Staubli VAL3: userPage.pjx

--- userPage.pjx ---
Parameters version=s7.5 stackSize=5000 millimeterUnit=true
Program file=changeTrsf.pgx
Program file=changeValue.pgx
Program file=clear.pgx
Program file=divideString.pgx
Program file=editNumField.pgx
Program file=findPos.pgx
Program file=getListPosition.pgx
Program file=getMenu.pgx
Program file=getView.pgx
Program file=insertDialog.pgx
Program file=isListEmpty.pgx
Program file=leftPos.pgx
Program file=listadd.pgx
Program file=listcreate.pgx
Program file=listcursor.pgx
Program file=listdel.pgx
Program file=listempty.pgx
Program file=listevent.pgx
Program file=listframe.pgx
Program file=listins.pgx
Program file=listredraw.pgx
Program file=listupdate.pgx
Program file=midPos.pgx
Program file=nullKey.pgx
Program file=numCopy.pgx
Program file=printScroll.pgx
Program file=questionDialog.pgx
Program file=read.pgx
Program file=rightPos.pgx
Program file=scroll.pgx
Program file=selectNewField.pgx
Program file=setCenter.pgx
Program file=setMenu.pgx
Program file=setSizeList.pgx
Program file=setView.pgx
Program file=showBoolStatus.pgx
Program file=strfill.pgx
Program file=strfillchr.pgx
Program file=stringCopy.pgx
Program file=stringToArray.pgx
Program file=stringToFxArray.pgx
Program file=strlength.pgx
Program file=timerDialog.pgx
Program file=type.pgx
Program file=typeCenter.pgx
Program file=typeLen.pgx
Program file=typeMenu.pgx
Program file=yes_no.pgx
Program file=yes_no_cancel.pgx
Data file=userPage.dtx

--- userPage.dtx ---
bool Show
bool bReadWrite = true
public bool bShowDialog
public bool bUseEscape
public bool bUseRefresh
public num nBottomX[2]
  [0] = 17
  [1] = 17
public num nBottomY = 11
num nFirst
num nKey
num nOffSet
num nOldValue[2]
  [0] = 200
  [1] = 200
public num nPage = 10
public num nTopX[2]
  [0] = 21
  [1] = 21
public num nTopY
public num nView
public string sItems = "home"
string sMessage[3]
  [0] = "VALPLAST QUITTING..."
  [1] = " "
  [2] = "PLEASE WAIT"
public string sTitle = "HOME"

--- changeTrsf.pgx ---
public program changeTrsf(trsf& x_tTrsf[], string x_sTitle, string x_sComment)
  local bool l_bRefresh
  local num l_nView
  local num l_nIndex
  local string l_sItem
  local trsf l_tTrsf
  local string l_sEvent
  local string l_sEmpty
  local num l_nAddon
begin
  //logMsg("[KERNEL] INTERFACE:PAGE changeTrsf "+x_sTitle)
  // INIT all
  l_bRefresh=false
  l_nIndex=0
  l_nView=0
  call setSizeList(19,0,19,8)
  call setView(false)
  l_tTrsf=x_tTrsf
  //release the button
  call nullKey(nKey)
  // set the frame
  do
    cls()
    call type(0,12,x_sComment)
    call typeMenu(8,"OK")
    call listcreate(x_sTitle)
    l_sItem=("coord  X > "+toString(".2",l_tTrsf.x))
    call listadd(l_sItem)
    l_sItem=("coord  Y > "+toString(".2",l_tTrsf.y))
    call listadd(l_sItem)
    l_sItem=("coord  Z > "+toString(".2",l_tTrsf.z))
    call listadd(l_sItem)
    l_sItem=("coord RX > "+toString(".2",l_tTrsf.rx))
    call listadd(l_sItem)
    l_sItem=("coord RY > "+toString(".2",l_tTrsf.ry))
    call listadd(l_sItem)
    l_sItem=("coord RZ > "+toString(".2",l_tTrsf.rz))
    call listadd(l_sItem)
    // show the list
    nView=l_nIndex
    call listupdate(l_nIndex-l_nView)
    do
      l_nView=nView
      nKey=get()
      //l_pPoint.trsf=l_tTrsf
      call listevent(nKey,l_nIndex,l_sEvent)
      switch nKey
        case 270
          //
          // clean the line
          call listcursor(nView,false)
          l_sEmpty=""
          switch l_nIndex
            case 0
              //  x-value
              call changeValue(l_tTrsf.x,0,0,10+40-nBottomX,nView+1,l_sEmpty)
            break
            case 1
              //  y-value
              call changeValue(l_tTrsf.y,0,0,10+40-nBottomX,nView+1,l_sEmpty)
            break
            case 2
              //  z-value
              call changeValue(l_tTrsf.z,0,0,10+40-nBottomX,nView+1,l_sEmpty)
            break
            case 3
              //  rx-value
              call changeValue(l_tTrsf.rx,0,0,10+40-nBottomX,nView+1,l_sEmpty)
            break
            case 4
              //  ry-value
              call changeValue(l_tTrsf.ry,0,0,10+40-nBottomX,nView+1,l_sEmpty)
            break
            case 5
              //  rz-value
              call changeValue(l_tTrsf.rz,0,0,10+40-nBottomX,nView+1,l_sEmpty)
            break
            case 6
              // addon
              l_nIndex=find(l_sEvent,">")
              call changeValue(l_nAddon,0,0,l_nIndex+1+2+nTopX,nView+nTopY+1,l_sEmpty)
            break
          endSwitch
          l_bRefresh=true
        break
        case 278
          // VALIDATE
          x_tTrsf=l_tTrsf
        break
      endSwitch
    until l_bRefresh==true or nKey==255 or nKey==278
    l_bRefresh=false
  until nKey==255 or nKey==278
  // check the key
  if nKey==278
    // validate
    x_tTrsf=l_tTrsf
  endIf
  // release the resource
  call nullKey(nKey)
end

--- changeValue.pgx ---
public program changeValue(num& x_nValue[], num x_nMin, num x_nMax, num x_nX, num x_nY, string& x_sItems[])
  local num l_nOldValue[2]
  local string l_sItem
  local string l_sMessage
  local bool l_bComma
  local string l_sEmpty
begin
  //---------------------------------
  // Staubli copyright 2005
  //                By toneage
  //[Public]-------------------------
  //
  // x_nValue:  num to change
  // x_nMax:    max value
  // x_nMin:    min value
  // x_nX:      X position
  // x_nY:      Y position
  // x_sItems   message
  //
  // look if the value is between max and min
  //
  if x_nMin>x_nMax
    return
  endIf
  //
  // print the line in white
  //
  // call listCleanLine()
  //
  call nullKey(nKey)
  l_nOldValue[1]=round(x_nValue)
  x_nValue=(round(x_nValue*100))/100
  l_nOldValue=x_nValue
  // check if is using the comma or not
  if l_nOldValue!=l_nOldValue[1]
    l_bComma=true
  else
    l_bComma=false
  endIf
  // start
  call clear(0,13)
  do
    if x_sItems==""
      //
      //  use the get num
      //
      if l_bComma
        call strfill(l_sEmpty,len(toString(".2",x_nValue)),l_sEmpty)
      else
        call strfill(l_sEmpty,len(toString("",x_nValue)),l_sEmpty)
      endIf
      call type(x_nX,x_nY,l_sEmpty)
      gotoxy(x_nX,x_nY)
      nKey=get(x_nValue)
      // check the comma again
      if round(x_nValue)!=x_nValue
        l_bComma=true
      endIf
      //
      // CHECK for MIN MAX VALUE
      //
      if x_nMax!=x_nMin or x_nMin!=0
        if x_nValue>x_nMax
          //
          // ask if you want to continue
          //
          popUpMsg("MAX: "+toString(".2",x_nMax))
          x_nValue=l_nOldValue
          //x_nValue=x_nMax
          nKey=-1
        else
          if x_nValue<x_nMin
            //
            popUpMsg("MIN: "+toString(".2",x_nMin))
            //x_nValue=x_nMin
            x_nValue=l_nOldValue
            nKey=-1
          endIf
        endIf
      endIf
      //
      // UPDATE THE VALUE
      //
      if l_bComma
        call type(x_nX,x_nY,toString(".2",x_nValue))
      else
        call type(x_nX,x_nY,toString("",x_nValue))
      endIf
    else
      //
      // STRING CHOICE
      //
      // show a list if there is the place
      call setSizeList(x_nX-1,max(0,x_nY-1),40-x_nX-1,min(13-x_nY,size(x_sItems)))
      call listcreate("")
      call listadd(x_sItems)
      call selectNewField(x_nValue,x_nValue,0)
      do
        nKey=get()
        call listevent(nKey,x_nValue,l_sItem)
      until nKey==270 or nKey==255
    endIf
  until nKey==270 or nKey==255
  if nKey==255
    bUseEscape=true
    x_nValue=l_nOldValue
    if x_sItems!=""
      x_sItems=x_sItems[l_nOldValue]
    endIf
  else
    bUseEscape=false
  endIf
end

--- clear.pgx ---
public program clear(num pX (dimensions=1), num pY (dimensions=1))
  local num i
  local num lLen
begin
  //---------------------------------
  //      C L E A R   L I N E
  //---------------------------------
  // Erase a pY line from the column
  // pX to end
  //
  //
  call typeLen(pX,pY," ",40-pX)
  gotoxy(pX,pY)
end

--- divideString.pgx ---
program divideString(string& x_sMsg[] (dimensions=1), num& x_nLine[] (dimensions=1))
  local string l_sCopyMsg
  local num l_nLength
  local string l_sSwap
  local num l_nFlag
  local num l_nTotalFlag
  local string l_sCR
  local num l_nPosCR
  local num i
begin
  //
  //  using:
  // x_sMessage->  the message you want print to video
  // x_nLine->     the number of the line that will be use
  //
  //
  // CARRIAGE RETURN
  l_sCR="#"
  x_nLine=0
  //length of a line for a message
  l_nLength=38
  // copy the msg
  l_sCopyMsg=x_sMsg
  // first case
  call findPos(l_sCopyMsg,l_sCR,l_nPosCR)
  if (getDisplayLen(l_sCopyMsg)>l_nLength-1) or (l_nPosCR!=-1)
    // compose the message
    do
      l_sSwap=l_sCopyMsg
      // set the x_sMsg
      if size(x_sMsg)-1<x_nLine
        append(x_sMsg)
      endIf
      call findPos(l_sCopyMsg,l_sCR,l_nPosCR)
      //
      if (getDisplayLen(l_sCopyMsg)>l_nLength-1 or (l_nPosCR!=-1)) and x_nLine<8
        // divide the string
        l_nTotalFlag=0
        call findPos(l_sCopyMsg,l_sCR,l_nPosCR)
        //
        // divide the string
        //
        if l_nPosCR!=-1 and l_nPosCR<l_nLength
          // CARRIAGE RETURN
          call leftPos(l_sCopyMsg,l_nPosCR,l_sSwap)
          //l_sSwap=left(l_sCopyMsg,l_nPosCR)
          call rightPos(l_sCopyMsg,getDisplayLen(l_sCopyMsg)-(l_nPosCR)-1,l_sCopyMsg)
          //l_sCopyMsg=right(l_sCopyMsg,len(l_sCopyMsg)-(l_nPosCR)-1)
          if getDisplayLen(l_sSwap)==0
            l_sSwap=" "
          endIf
        else
          //
          // search for the space then return
          //
          do
            call findPos(l_sSwap," ",l_nFlag)
            //l_nFlag=find(l_sSwap," ")
            if l_nFlag!=-1 and l_nFlag<=l_nLength
              //l_sSwap=right(l_sSwap,len(l_sSwap)-l_nFlag-1)
              call rightPos(l_sSwap,getDisplayLen(l_sSwap)-l_nFlag-1,l_sSwap)
              l_nTotalFlag=l_nTotalFlag+l_nFlag+1
            else
              if l_nTotalFlag==0 and (l_nFlag==-1 or l_nFlag>l_nLength)
                l_nFlag=-1
                l_nTotalFlag=38
              endIf
            endIf
          until l_nTotalFlag>=l_nLength+2 or l_nFlag==-1
          // NORMAL
          if l_nTotalFlag==0
            // FULL LINE
            call leftPos(l_sCopyMsg,l_nLength,l_sSwap)
            //l_sSwap=left(l_sCopyMsg,l_nLength)
            //l_sCopyMsg=right(l_sCopyMsg,len(l_sCopyMsg)-l_nLength)
            call rightPos(l_sCopyMsg,getDisplayLen(l_sCopyMsg)-l_nLength,l_sCopyMsg)
          else
            // DIVIDE IT
            call leftPos(l_sCopyMsg,l_nTotalFlag-l_nFlag-2,l_sSwap)
            //l_sSwap=left(l_sCopyMsg,l_nTotalFlag-l_nFlag-2)
            //l_sCopyMsg=right(l_sCopyMsg,len(l_sCopyMsg)-(l_nTotalFlag-l_nFlag-1))
            call rightPos(l_sCopyMsg,getDisplayLen(l_sCopyMsg)-(l_nTotalFlag-l_nFlag-1),l_sCopyMsg)
          endIf
        endIf
        // set the string
        x_sMsg[x_nLine]=l_sSwap
        x_nLine=x_nLine+1
      else
        // limit the string
        call rightPos(l_sSwap,l_nLength,x_sMsg[x_nLine])
        //x_sMsg[x_nLine]=right(l_sSwap,l_nLength)
        l_sSwap=""
      endIf
    until l_sSwap==""
  endIf
end

--- editNumField.pgx ---
public program editNumField(string x_sTitle, string& x_sItemName[], num& x_nItem[], num& x_nMin[], num& x_nMax[])
  local num j
  local num l_nSize
  local num l_nKey
  local string l_sEvent
  local num l_nIndex
  local num l_nField
  local string l_sItem
  local num i
  local string l_sEmpty
begin
  //
  // clear & copy
  //
  // nView=nFirst=0
  //call listempty()
  call numCopy(x_nItem,nOldValue)
  call numCopy(x_nItem,nOffSet)
  for j=0 to size(nOffSet)-1
    nOffSet[j]=0
  endFor
  // take the size
  l_nSize=size(x_nItem)-1
  // create the LIST
  call setSizeList(2,max((6-l_nSize/2)-2,2),34,min((l_nSize+1),8))
  call listcreate(x_sTitle)
  //
  // insert items
  //
  for j=0 to l_nSize
    l_sItem=x_sItemName[j]
    if l_sItem!=""
      call strlength(l_sItem,26)
      l_sItem=l_sItem+": "+toString(".1",x_nItem[j])
      call listadd(l_sItem)
      nOffSet[j]=nOffSet[max(j-1,0)]
    else
      nOffSet[j]=nOffSet[max(j-1,0)]+1
    endIf
  endFor
  // update the list
  call listupdate(0)
  do
    call clear(0,13)
    call typeMenu(8,"OK")
    l_nKey=get()
    call listevent(l_nKey,l_nIndex,l_sEvent)
    // use the offset
    i=l_nIndex+nOffSet[max(l_nIndex,0)]
    // on Enter Key
    if l_nKey==270
      call listcursor(l_nIndex,false)
      if size(x_nMin)==size(x_nItem)
        // use min and max
        l_sEmpty=""
        call changeValue(x_nItem[i],x_nMin[i],x_nMax[i],31,nView+nTopY+1,l_sEmpty)
      else
        call changeValue(x_nItem[i],x_nMin,x_nMax,31,nView+nTopY+1,l_sEmpty)
      endIf
      // UPDATE
      call listdel(l_nIndex)
      l_sItem=x_sItemName[i]
      call strlength(l_sItem,26)
      l_sItem=l_sItem+": "+toString(".1",x_nItem[i])
      call listins(l_sItem,l_nIndex)
      call listupdate(l_nIndex-nView)
    endIf
  until l_nKey==278 or l_nKey==255
  // escape use ?
  if l_nKey==255
    bUseEscape=true
    call numCopy(nOldValue,x_nItem)
  else
    bUseEscape=false
  endIf
  // exit
  call nullKey(l_nKey)
end

--- findPos.pgx ---
public program findPos(string x_sItem1 (dimensions=1), string x_sItem2 (dimensions=1), num& x_nPos[] (dimensions=1))
  local num l_nPos
begin
  // find the char using getDisplayLen
  l_nPos=find(x_sItem1,x_sItem2)
  if l_nPos!=-1
    x_nPos=getDisplayLen(left(x_sItem1,l_nPos))
  else
    x_nPos=-1
  endIf
end

--- getListPosition.pgx ---
public program getListPosition(num& x_nIndexX[] (dimensions=1), num& x_nIndexY[] (dimensions=1))
begin
  x_nIndexX=nTopX+1
  x_nIndexY=nFirst+nView+nTopY+1
end

--- getMenu.pgx ---
public program getMenu(string& x_sMenu[] (dimensions=1), bool& x_bUseMenu[] (dimensions=1))
// set the function button using the menu string
  local num i
begin
  //
  // STAUBLI Application
  // set the x_bUseMenu using the Menu
  // array string
  //
  for i=0 to (size(x_bUseMenu)-1)
    x_bUseMenu[i]=false
    if (size(x_sMenu)-1)>=i
      if x_sMenu[i]!=""
        // active the button
        x_bUseMenu[i]=true
      endIf
    endIf
  endFor
end

--- getView.pgx ---
public program getView(bool& x_bView[] (dimensions=1))
begin
  if nBottomX==38
    x_bView=true
  else
    x_bView=false
  endIf
end

--- insertDialog.pgx ---
public program insertDialog(string x_sMsg, num& x_nItem[], num x_nMin, num x_nMax)
  local num l_nStartLine
  local num l_nLine
  local num i
  local num l_nPX
  local num l_nPY
  local string l_sItem
  local string l_sMessage
  local string l_sEmpty
begin
  //
  // modify the x_sItem, using a min max range
  //
  if watch(bShowDialog==false,3)==false
    bShowDialog=false
    return
  else
    setMutex(bShowDialog)
    // clear the line
    call clear(0,13)
    // look for the comma
    if round(x_nItem)!=x_nItem
      l_sItem=toString(".2",x_nItem)
    else
      l_sItem=toString("",x_nItem)
    endIf
    // print the line
    l_sItem=x_sMsg+">"+l_sItem
    call stringCopy(l_sItem,sMessage)
    // divide the sentence
    call divideString(sMessage,l_nLine)
    l_nStartLine=round(5-l_nLine/2)
    // Start LINE
    call type(0,l_nStartLine-2,"┌──────────────────────────────────────┐")
    call type(0,l_nStartLine-1,"│                                      │")
    // write the message
    for i=0 to l_nLine
      //call type(,"                                      ")
      l_sMessage=sMessage[i]
      call typeCenter(i+l_nStartLine,l_sMessage,38,false)
      call type(0,l_nStartLine+i,"│"+l_sMessage+"│")
    endFor
    // end LINE
    call type(0,l_nStartLine+l_nLine+1,"│                                      │")
    call type(0,l_nStartLine+l_nLine+2,"└──────────────────────────────────────┘")
    l_nPX=find(l_sMessage,">")+2
    l_nPY=l_nStartLine+l_nLine
    // change the value
    call changeValue(x_nItem,x_nMin,x_nMax,l_nPX,l_nPY,l_sEmpty)
    //
    bShowDialog=false
    bUseRefresh=true
    //
  endIf
end

--- isListEmpty.pgx ---
public program isListEmpty(bool& x_bEmpty[] (dimensions=1))
begin
  if size(sItems)==1 and sItems[0]==""
    x_bEmpty=true
  else
    x_bEmpty=false
  endIf
end

--- leftPos.pgx ---
public program leftPos(string x_sItem (dimensions=1), num x_nLength (dimensions=1), string& x_sResult[] (dimensions=1))
  local num i
  local num l_nLength
  local string l_sItem
begin
  //
  l_sItem=x_sItem
  //
  if len(l_sItem)!=getDisplayLen(l_sItem) and x_nLength>0
    for i=0 to len(x_sItem)-1
      l_nLength=l_nLength+getDisplayLen(left(l_sItem,1))
      l_sItem=right(l_sItem,len(l_sItem)-1)
      if l_nLength==x_nLength
        x_sResult=left(x_sItem,i+1)
        return
      else
        if l_nLength>x_nLength
          x_sResult=left(x_sItem,i)
          return
        endIf
      endIf
    endFor
    // else
  endIf
  x_sResult=left(x_sItem,max(x_nLength,0))
  // endIf
end

--- listadd.pgx ---
public program listadd(string& x_sItems[] (dimensions=1))
  local num i
  local num l_nSize
begin
  //---------------------------------
  // insert x_sItems into the list
  //---------------------------------
  //
  // x_sItems:      Items to add
  //
  //---------------------------------
  // Staubli copyright 2005
  //                By toneage
  //[Public]-------------------------
  //
  //
  for i=0 to (size(x_sItems)-1)
    if (size(sItems)!=1 or sItems!="") and x_sItems[i]!=""
      insert(sItems[size(sItems)])
      insert(bReadWrite[size(bReadWrite)])
    endIf
    if x_sItems[i]!=""
      sItems[size(sItems)-1]=x_sItems[i]
      // for default the RW is true
      bReadWrite[size(bReadWrite)-1]=true
    endIf
  endFor
end

--- listcreate.pgx ---
public program listcreate(string x_sTitle)
begin
  //
  // Staubli Copyright 2003 07 31
  //
  sTitle=x_sTitle
  call listframe(sTitle,nTopX,nTopY,nBottomX,nBottomY)
  call listempty()

end

--- listcursor.pgx ---
public program listcursor(num pView (dimensions=1), bool pShow (dimensions=1))
  local num lX
  local num lY
  local string message
  local bool l_bEmpty
begin
  //
  // toneage Staubli Copyright 2005
  //
  call isListEmpty(l_bEmpty)
  if !l_bEmpty
    nView=pView
    lX=nTopX+1
    lY=nTopY+1+pView
    if (nView+nFirst)>(size(sItems)-1)
      call strfill(sItems[size(sItems)-1],nBottomX,message)
    else
      call strfill(sItems[max(0,nView+nFirst)],nBottomX,message)
    endIf
    gotoxy(lX,lY)
    if (pShow==true)
      setTextMode(1)
      put(message)
      setTextMode(0)
    else
      setTextMode(0)
      put(message)
    endIf
  endIf
end

--- listdel.pgx ---
public program listdel(num x_nIndex (dimensions=1))
  local num l_nSize
begin
  //
  // Staubli Copyright 2005 toneage
  //
  l_nSize=size(sItems)-1
  if ((x_nIndex>=0) and (x_nIndex<=l_nSize))
    if l_nSize>0
      delete(sItems[x_nIndex])
      delete(bReadWrite[x_nIndex])
    else
      sItems=""
      bReadWrite=true
    endIf
  endIf
end

--- listempty.pgx ---
public program listempty()
  local num lI
  local num lLen
  local string lRun[5]
  local num lRuni
begin
  //
  // Staubli Copyright 2003 06 20
  //
  lLen=size(sItems)-1
  for lI=0 to lLen
    if lI>0
      delete(sItems[0])
      delete(bReadWrite[0])
    endIf
  endFor
  sItems=""
  //
end

--- listevent.pgx ---
public program listevent(num pkey (dimensions=1), num& pIndex[] (dimensions=1), string& pItem[] (dimensions=1))
  local num lVal
  local num l_nSize
  local bool l_bEmpty
begin
  //
  // Toneage Staubli product
  //
  //
  // get the item in the list and scroll it
  //
  call isListEmpty(l_bEmpty)
  // not allowed negative value
  nView=max(0,nView)
  nFirst=max(0,nFirst)
  pIndex=max(0,pIndex)
  // look for the empty
  if !l_bEmpty
    l_nSize=size(sItems)-1
    // check the overFlow
    l_nSize=size(sItems)-1
    if (nFirst+nView>l_nSize)
      // reset the value
      nFirst=nView=0
    endIf
    // security...
    switch (pkey)
      //Up
      case 261
        if ((nView-1)>=0)
          // no need to scroll only change cursor position
          call listcursor(nView,false)
          nView=nView-1
          call listcursor(nView,true)
          // print the scroll
          //call printScroll()
        else
          if nView==0
            // scroll up
            if ((nFirst-1)>=0)
              nFirst=nFirst-1
              call listupdate(nFirst)
            else
              // go to the end
              if nView+nFirst!=l_nSize
                call listcursor(nView,false)
                call selectNewField(l_nSize,nFirst+nView,nView)
              endIf
            endIf
          endIf
        endIf
      break
      //Down
      case 266
        if ((nView+nFirst+1)<size(sItems))
          // no need to scroll only chenge cursor position
          if ((nView+1)<nBottomY)
            call listcursor(nView,false)
            nView=nView+1
            call listcursor(nView,true)
            // print the scroll
            //call printScroll()
          else
            // move UP
            nFirst=nFirst+1
            call listupdate(nFirst)
          endIf
        else
          // go to the top
          if !(nView==0 and nFirst==0)
            call listcursor(nView,false)
            nView=0
            call listupdate(0)
          endIf
        endIf
      break
      //Page Up
      case 262
        if !(nView==0 and nFirst==0)
          call listcursor(nView,false)
          if ((nFirst+nView-nBottomY)>=0)
            // move one page up
            call selectNewField(nFirst+nView-nBottomY,nFirst+nView,nView)
          else
            // go to home
            nView=0
            call listupdate(0)
          endIf
        endIf
      break
      //Page Down
      case 267
        if nView+nFirst!=l_nSize
          call listcursor(nView,false)
          if ((nView+nFirst+nBottomY)<size(sItems)-1)
            // move one page down
            call selectNewField(nFirst+nView+nBottomY,nFirst+nView,nView)
          else
            // go to the end
            call selectNewField(l_nSize,nFirst+nView,nView)
          endIf
        endIf
      break
      //End
      case 269
        if nView+nFirst!=l_nSize
          // move to end
          call listcursor(nView,false)
          call selectNewField(l_nSize,nFirst+nView,nView)
        endIf
      break
      //Home
      case 265
        if !(nView==0 and nFirst==0)
          // move to home
          call listcursor(nView,false)
          nView=0
          call listupdate(0)
        endIf
      break
      default
      break
    endSwitch
    pIndex=nFirst+nView
    pItem=sItems[pIndex]
    //
  else
    // reset the item
    pItem=""
    pIndex=0
  endIf
end

--- listframe.pgx ---
program listframe(string pTitle (dimensions=1), num pX (dimensions=1), num pY (dimensions=1), num pDx (dimensions=1), num pDy (dimensions=1))
  local num lDx
  local num lDy
  local num lI
  local num lJ
  local string lStr
  local string lStrLine
  local num lValue
begin
  //
  // Staubli Copyright 2003 06 20
  //
  lStrLine="─────────────────────────────────────────"
  lDx=pDx
  lDy=pDy
  //Top
  lStr="┌"+mid(lStrLine,lDx,0)+"┐"
  gotoxy(pX,pY)
  put(lStr)
  lValue=pX+2
  //Title
  if pTitle!=""
    call leftPos("┤"+pTitle+"│",lDx+1,pTitle)
    gotoxy(pX+lDx-getDisplayLen(pTitle)+2,pY)
    put(pTitle)
  endIf
  //Containt
  for lJ=1 to lDy
    lValue=pY+lJ
    lStr="│"
    gotoxy(pX,lValue)
    put(lStr)
    gotoxy(pX+lDx+1,lValue)
    put(lStr)
  endFor
  //Bottom
  lValue=pY+lJ
  lStr="└"+mid(lStrLine,lDx,0)+"┘"
  gotoxy(pX,lValue)
  put(lStr)
end

--- listins.pgx ---
public program listins(string& x_sItems[] (dimensions=1), num x_nPos (dimensions=1))
  local num i
  local num l_nSize
begin
  //
  // Staubli Copyright 2005
  //
  l_nSize=size(sItems)-1
  if ((x_nPos>=0) and (x_nPos<=l_nSize))
    for i=0 to (size(x_sItems)-1)
      if size(sItems)!=1 or sItems!=""
        insert(sItems[x_nPos+i])
        insert(bReadWrite[x_nPos+i])
      endIf
      sItems[x_nPos+i]=x_sItems[i]
      // for default the RW is true
      bReadWrite[x_nPos+i]=true
    endFor
  else
    call listadd(x_sItems)
  endIf
end

--- listredraw.pgx ---
public program listredraw(num pFirst (dimensions=1))
begin
  //
  // Staubli Copyright 2003 06 20
  //
  call listframe(sTitle,nTopX,nTopY,nBottomX,nBottomY)
  call listupdate(pFirst)
end

--- listupdate.pgx ---
public program listupdate(num pFirst)
  local num lI
  local num lLen
  local string lStr
  local string lStr2
  local num lValue
  local num lView
  local num lX
  local num lY
  local num l_nSize
  local bool l_bEmpty
begin
  //
  // insert into the box all the data
  //
  // to prevent a negative value
  if pFirst>0
    nFirst=pFirst
  else
    nFirst=0
  endIf
  // save the coordinate
  lValue=nBottomY-1
  // check the overFlow
  l_nSize=size(sItems)-1
  if (nFirst+nView>l_nSize)
    // reset the value
    nFirst=nView=0
  endIf
  lI=0
  // check the unKnow poblem
  if l_nSize<lValue
    if nFirst!=0
      nView=nView+nFirst
      nFirst=0
    endIf
  endIf
  do
    lX=nTopX+1
    lY=nBottomY+lI-1
    lY=nTopY+lI+1
    lLen=nBottomX
    if ((lI+nFirst)<size(sItems))
      // print the item
      if (l_nSize>=0)
        lStr=mid(sItems[(lI+nFirst)],lLen,0)
      endIf
    else
      // print the blank line
      lStr="                                        "
    endIf
    // fill the line
    call strfill(lStr,lLen,lStr2)
    gotoxy(lX,lY)
    put(lStr2)
    lI=lI+1
  until (lI>lValue)
  // underlien the actual line
  call isListEmpty(l_bEmpty)
  if !l_bEmpty
    call listcursor(nView,true)
  else
    call listcursor(nView,false)
    nView=0
    nFirst=0
  endIf
  // print the scroll
  call printScroll()
end

--- midPos.pgx ---
public program midPos(string x_sItem (dimensions=1), num x_nLenght (dimensions=1), num x_nPos (dimensions=1), string& x_sResult[] (dimensions=1))
  local string l_sLeft
begin
  // LEFT SIDE
  call leftPos(x_sItem,x_nLenght+x_nPos,l_sLeft)
  // update
  x_sResult=l_sLeft
  // RIGHT SIDE
  call rightPos(l_sLeft,x_nLenght,x_sResult)
  // OK ....
end

--- nullKey.pgx ---
public program nullKey(num& x_nKey[])
begin
  wait(getKey()==-1)
  x_nKey=0
end

--- numCopy.pgx ---
public program numCopy(num& x_nCopy[] (dimensions=1), num& x_nPaste[] (dimensions=1))
// Copy all the value from the x_nCopy to x_nPaste
  local num i
  local num l_nSize
begin
  // Copy all the value from the first element to the second one
  //
  // redim the Paste String ARRAY
  //
  if size(x_nPaste)!=size(x_nCopy)
    resize(x_nPaste,1,size(x_nCopy))
  endIf
  // COPY ALL THE FIELD
  for i=0 to (size(x_nCopy)-1)
    x_nPaste[i]=x_nCopy[i]
  endFor
end

--- printScroll.pgx ---
program printScroll()
  local num i
  local num lX
  local num lY
begin
  //
  // put the scroll
  //
  //if size(sItems)>nBottomY
  // find the percentage
  //windows style
  //i=(size(sItems)-nBottomY+1)/(nFirst+1)
  // nokia style
  i=(size(sItems))/(nFirst+nView+1)
  lX=nTopX+nBottomX+1
  lY=roundUp((nBottomY)/i+nTopY)
  for i=nTopY+1 to nBottomY
    gotoxy(lX,i)
    if (i==nTopY+1 and nFirst!=0)or(i==nBottomY and nFirst<=size(sItems)-1-(nBottomY-nTopY))and size(sItems)>nBottomY
      // show more items
      put("+")
    else
      put("│")
    endIf
  endFor
  //endIf
end

--- questionDialog.pgx ---
public program questionDialog(string x_sMsg, string& x_sButton[], num& x_nResult[])
  local bool lExit
  local num nLine
  local num i
  local num nStartLine
  local string l_sMessage
begin
  //---------------------------------
  //      D I A L O G    B O X
  //---------------------------------
  //
  // Show one dialog box. with an confirm question
  //
  if watch(bShowDialog==false,3)==false
    bShowDialog=false
    return
  else
    setMutex(bShowDialog)
    //
    //
    if x_sMsg!=""
      call stringCopy(x_sMsg,sMessage)
      call divideString(sMessage,nLine)
      nStartLine=round(5-nLine/2)
      // Start LINE
      call type(0,nStartLine-2,"┌──────────────────────────────────────┐")
      call type(0,nStartLine-1,"│                                      │")
      // write the message
      for i=0 to nLine
        l_sMessage=sMessage[i]
        call typeCenter(i+nStartLine,l_sMessage,38,false)
        call type(0,nStartLine+i,"│"+l_sMessage+"│")
      endFor
      // end LINE
      call type(0,nStartLine+nLine+1,"│                                      │")
      call type(0,nStartLine+nLine+2,"└──────────────────────────────────────┘")
    endIf
    // write the button message
    call clear(0,13)
    for i=0 to size(x_sButton)-1
      call typeMenu(8-i,x_sButton[i])
    endFor
    lExit=false
    x_nResult=-100
    do
      nKey=get()
      switch (nKey)
        case 270
          x_nResult=0
        break
        case 255
          x_nResult=-1
          bUseEscape=true
        break
        default
          // look if the button press is defined
          if (nKey>=271 and nKey<=278) and ((279-nKey)<=size(x_sButton))
            if x_sButton[278-nKey]!=""
              x_nResult=279-nKey
            endIf
          endIf
        break
      endSwitch
    until (x_nResult!=-100)
    //
    call nullKey(nKey)
    if x_nResult!=-1
      bUseEscape=false
    endIf
    //
    // release
    bShowDialog=false
    bUseRefresh=true
  endIf
end

--- read.pgx ---
public program read(num pX (dimensions=1), num pY (dimensions=1), string& pMsg[] (dimensions=1), num pLen (dimensions=1), bool pCrypt (dimensions=1))
  local num lLen
  local bool lExit
  local bool lBlk
  local num l
  local num p
  local num lTps
  local string lMsg
  local string lView
  local string lStr
begin
  //---------------------------------
  //  R E A D   O N E   S T R I N G
  //---------------------------------
  // Read one string from the pX
  // column and pY line
  //
  lTps=clock()
  lMsg=pMsg
  p=len(lMsg)
  // cryptage
  if pCrypt
    do
      l=len(lMsg)
      nKey=getKey()
      if ((clock()-lTps)>=0.5)
        if lBlk==true
          lBlk=false
        else
          lBlk=true
        endIf
        lTps=clock()
      endIf
      if (nKey>=32) and (nKey<=126)
        if ((len(lMsg)+1)<=pLen)
          lMsg=lMsg+chr(nKey)
        endIf
      else
        if (nKey==263) and (len(lMsg)>0)
          lMsg=mid(lMsg,len(lMsg)-1,0)
        endIf
      endIf
      if (lStr!=lMsg)
        call strfillchr(lMsg,lView,"*")
        lStr=lMsg
      endIf
      if lBlk==true
        call typeLen(pX,pY,lView+"|",pLen+1)
      else
        call typeLen(pX,pY,lView+" ",pLen+1)
      endIf
      //
      // release the resource
      delay(0)
    until (nKey==270) or (nKey==255)
  else
    // normal read
    // delete the old value
    setTextMode(0)
    call strfillchr(lMsg,lView," ")
    call typeLen(pX,pY,lView,40-pX-1)
    // read the new one
    gotoxy(pX,pY)
    get(lMsg)
  endIf
  // result
  if isKeyPressed(270) or lMsg!=""
    pMsg=lMsg
  endIf
  if isKeyPressed(255)
    bUseEscape=true
  else
    bUseEscape=false
  endIf
end

--- rightPos.pgx ---
public program rightPos(string x_sItem (dimensions=1), num x_nLength (dimensions=1), string& x_sResult[] (dimensions=1))
  local num i
  local num l_nLength
  local string l_sItem
begin
  //
  l_sItem=x_sItem
  // divide the string...
  if len(l_sItem)!=getDisplayLen(l_sItem) and x_nLength<=getDisplayLen(l_sItem) and x_nLength>0
    for i=len(x_sItem)-1 to 0 step -1
      l_nLength=l_nLength+getDisplayLen(right(l_sItem,1))
      l_sItem=left(l_sItem,len(l_sItem)-1)
      if l_nLength==x_nLength
        x_sResult=right(x_sItem,len(x_sItem)-i)
        return
      else
        if l_nLength>x_nLength
          x_sResult=right(x_sItem,len(x_sItem)-i-1)
          return
        endIf
      endIf
    endFor
  endIf
  //else
  x_sResult=right(x_sItem,max(x_nLength,0))
  //endIf
end

--- scroll.pgx ---
public program scroll(num x_nX (dimensions=1), num x_nY (dimensions=1), num x_nDim (dimensions=1), num x_nPos (dimensions=1))
// create a scroll bar
  local string l_sMessage
  local string l_sLine
  local num l_nPos
  local string l_sScrool
begin
  // use the scroll
  if x_nPos>0 and x_nPos<=100
    l_nPos=round(x_nDim*x_nPos/100)
    if l_nPos>0
      // make the scroll
      call strfill(l_sScrool,l_nPos,l_sScrool)
      call strfillchr(l_sScrool,l_sScrool,"■")
    endIf
    // make the line
    call strfill(l_sLine,x_nDim-l_nPos,l_sLine)
    call strfillchr(l_sLine,l_sLine,"─")
    l_sMessage="└"+l_sScrool+l_sLine+"┘"
    // show the line
    call type(x_nX,x_nY,l_sMessage)
  endIf
end

--- selectNewField.pgx ---
public program selectNewField(num x_nSelected (dimensions=1), num x_nIndex (dimensions=1), num x_nView (dimensions=1))
  local num l_nFirst
begin
  //
  // SELECT THE NEW ITEM WITH A USER FRIENDLY SYSTEM
  //
  //NB -Selected  is the position of the new item
  //   -Index     is the current position
  //   -nView     is the current position relative to the screen depth
  // START
  //
  l_nFirst=max(x_nIndex-x_nView,0)
  if (x_nSelected==-1)
    nView=x_nView
    call listupdate(x_nIndex-x_nView)
  else
    //
    //  select the new field
    //
    // the new value is not in the screen
    if x_nSelected<=l_nFirst or abs(x_nSelected-l_nFirst)>=(nBottomY)
      // start from the beginnnig
      if x_nSelected<=l_nFirst and x_nSelected<nBottomY
        nView=x_nSelected
        call listupdate(0)
      else
        if x_nSelected<size(sItems)-nBottomY
          // move the list and select the field in the middle
          nView=roundUp(nBottomY/2)
        else
          nView=x_nSelected-(size(sItems)-nBottomY)
        endIf
        call listupdate(abs(x_nSelected-nView))
      endIf
    else
      // move only the nView of the field
      nView=abs(x_nSelected-l_nFirst)
      call listupdate(abs(x_nIndex-x_nView))
    endIf
  endIf
end

--- setCenter.pgx ---
program setCenter()
begin
end

--- setMenu.pgx ---
public program setMenu(string& x_sMenuName[] (dimensions=1), bool x_bShowName (dimensions=1), num x_nY (dimensions=1))
// Show the
  local num i
begin
  //
  // usage
  // menuname"choice1,choise2,..choise7,choice8"
  //
  // the page will start from the y- line
  //
  //
  if size(x_sMenuName)<10
    for i=0 to (size(x_sMenuName)-1)
      if x_sMenuName[i]!="" and x_sMenuName[i]!=" "
        if x_bShowName==false
          call typeMenu(i+1,"F"+toString("1",i+1))
        else
          call typeMenu(i+1,x_sMenuName[i])
        endIf
        if x_nY!=-1
          call type(0,i+x_nY,("F"+(toString("1",i+1)+" "+x_sMenuName[i])))
        endIf
      endIf
    endFor
  endIf
end

--- setSizeList.pgx ---
public program setSizeList(num nPx (dimensions=1), num nPy (dimensions=1), num nPBottomX (dimensions=1), num nPBottomY (dimensions=1))
begin
  nTopX=nTopX[1]=nPx
  nTopY=nPy
  nBottomX=nBottomX[1]=nPBottomX
  nBottomY=nPBottomY
end

--- setView.pgx ---
public program setView(bool x_bLarge (dimensions=1))
begin
  // look if to enlarge the screen
  if x_bLarge
    nTopX[1]=nTopX
    nTopX=0
    nBottomX[1]=nBottomX
    nBottomX=38
  else
    nTopX=nTopX[1]
    nBottomX=nBottomX[1]
  endIf
  bUseRefresh=true
end

--- showBoolStatus.pgx ---
public program showBoolStatus(bool x_bStatus (dimensions=1), string& x_sEvent[] (dimensions=1))
begin
  if x_bStatus
    x_sEvent="[x]"
  else
    x_sEvent="[ ]"
  endIf
end

--- strfill.pgx ---
public program strfill(string pStrIn (dimensions=1), num pLenStrOut (dimensions=1), string& pStrOut[] (dimensions=1))
  local string lEmpty
  local num lLen
begin
  //---------------------------------
  //  F I L L   O N E   S T R I N G
  //---------------------------------
  // To fill the string with space
  // character
  //
  // look for asian message
  if getDisplayLen(pStrIn)<pLenStrOut
    // insert some space
    lEmpty="                                        "
    pStrOut=pStrIn
    lLen=(pLenStrOut-getDisplayLen(pStrIn))
    call midPos(lEmpty,lLen,0,pStrIn)
    pStrOut=pStrOut+pStrIn
  else
    if getDisplayLen(pStrIn)>pLenStrOut
      // divide the string
      call midPos(pStrIn,pLenStrOut,0,pStrOut)
    else
      // they are the same
      pStrOut=pStrIn
    endIf
  endIf
end

--- strfillchr.pgx ---
public program strfillchr(string pStrIn (dimensions=1), string& pStrOut[] (dimensions=1), string pChar (dimensions=1))
  local num lIndex
begin
  //---------------------------------
  //  F I L L   O N E   S T R I N G
  //---------------------------------
  // To fill the string with custom
  // character
  //
  //
  pStrOut=""
  if getDisplayLen(pStrIn)>0
    for lIndex=0 to (getDisplayLen(pStrIn)-1)
      pStrOut=pStrOut+pChar
    endFor
  endIf
end

--- stringCopy.pgx ---
public program stringCopy(string& x_sCopy[] (dimensions=1), string& x_sPaste[] (dimensions=1))
// Copy all the value from the x_sCopy to x_sPaste
  local num i
  local num l_nSize
begin
  // Copy all the value from the first element to the second one
  //
  // redim the Paste String ARRAY
  //
  //l_nSize=size(x_sPaste)
  if size(x_sPaste)!=size(x_sCopy)
    resize(x_sPaste,1,size(x_sCopy))
  endIf
  //  if size(x_sCopy)>size(x_sPaste)
  //    for i=l_nSize to (size(x_sCopy)-1)
  //      insert(x_sPaste[i])
  //    endFor
  //  else
  //    if size(x_sCopy)<size(x_sPaste)
  //      for i=size(x_sCopy) to l_nSize-1
  //        delete(x_sPaste[size(x_sCopy)])
  //      endFor
  //    endIf
  //  endIf
  // COPY ALL THE FIELD
  for i=0 to (size(x_sCopy)-1)
    x_sPaste[i]=x_sCopy[i]
  endFor
end

--- stringToArray.pgx ---
public program stringToArray(string x_sString (dimensions=1), string& x_sArray[] (dimensions=1))
// copy one String into an ARRAY of String
  local num i
  local num l_nItem
  local string l_sChar
  local string l_sEmpty
begin
  // define the char use to divide the items
  // PRIORITY
  //  ^
  //  ;
  //  ,
  //
  if find(x_sString,"^")==-1
    if find(x_sString,";")==-1
      l_sChar=","
    else
      l_sChar=";"
    endIf
  else
    l_sChar="^"
  endIf
  // init the X_sArray
  l_sEmpty=""
  call stringCopy(l_sEmpty,x_sArray)
  l_nItem=0
  do
    // increase the ARRAY SIZE
    if l_nItem>0
      insert(x_sArray[l_nItem])
    endIf
    i=find(x_sString,l_sChar)
    // look if was found
    if i!=-1
      // PUT INSIDE THE ARRAY THE STRING
      x_sArray[l_nItem]=left(x_sString,i)
      x_sString=delete(x_sString,i+1,0)
    else
      // look if is empty or not
      if len(x_sString)>0
        x_sArray[l_nItem]=(x_sString)
      endIf
    endIf
    l_nItem=l_nItem+1
  until i==-1
end

--- stringToFxArray.pgx ---
public program stringToFxArray(string x_sString (dimensions=1), string& x_sArray[] (dimensions=1))
// copy one String into an ARRAY of String
  local num i
  local num l_nItem
  local string l_sChar
  local string l_sEmpty
begin
  // define the char use to divide the items
  // PRIORITY
  //  ^
  //  ;
  //  ,
  //
  if find(x_sString,"^")==-1
    if find(x_sString,";")==-1
      l_sChar=","
    else
      l_sChar=";"
    endIf
  else
    l_sChar="^"
  endIf
  // init the X_sArray
  l_nItem=0
  do
    i=find(x_sString,l_sChar)
    // look if was found
    if i!=-1
      // PUT INSIDE THE ARRAY THE STRING
      x_sArray[l_nItem]=left(x_sString,i)
      x_sString=delete(x_sString,i+1,0)
    else
      // look if is empty or not
      if len(x_sString)>0
        x_sArray[l_nItem]=(x_sString)
      else
        x_sArray[l_nItem]=""
      endIf
    endIf
    l_nItem=l_nItem+1
  until i==-1
  // fill with empty field for the rest
  for i=l_nItem to size(x_sArray)-1 step 1
    x_sArray[i]=""
  endFor
end

--- strlength.pgx ---
public program strlength(string& pStr[] (dimensions=1), num pLen (dimensions=1))
  local string lStrEmpty
  local string l_sTemp
begin
  lStrEmpty="                                        "
  // look for asian message
  if getDisplayLen(pStr)>pLen and pLen>0
    // need to divide the message
    if getDisplayLen(pStr)==len(pStr)
      if mid(pStr,1,pLen)!=" "
        // european message
        pStr=mid(pStr,pLen-1,0)
        pStr=pStr+"."
      else
        // found and empty space
        pStr=mid(pStr,pLen,0)
      endIf
    else
      // asian one
      call midPos(pStr,pLen,0,pStr)
    endIf
  else
    if getDisplayLen(pStr)<pLen
      // european
      if getDisplayLen(pStr)==len(pStr)
        pStr=pStr+mid(lStrEmpty,pLen-getDisplayLen(pStr),0)
      else
        // asian
        call midPos(lStrEmpty,pLen-getDisplayLen(pStr),0,l_sTemp)
        pStr=pStr+l_sTemp
      endIf
    else
      // they are the same
      //
    endIf
  endIf
end

--- timerDialog.pgx ---
public program timerDialog(string x_sMsg, num x_nTime)
  local num l_nTime
  local num l_nStartLine
  local num l_nLine
  local num i
  local string l_sMessage
begin
  //
  // use for other task
  //
  if watch(bShowDialog==false,3)==false
    bShowDialog=false
    return
  else
    setMutex(bShowDialog)
    //
    //call listempty()
    //
    l_nTime=clock()
    call stringCopy(x_sMsg,sMessage)
    call divideString(sMessage,l_nLine)
    l_nStartLine=round(5-l_nLine/2)
    do
      // Start LINE
      call type(0,l_nStartLine-2,"┌──────────────────────────────────────┐")
      call type(0,l_nStartLine-1,"│                                      │")
      // write the message
      for i=0 to l_nLine
        call type(0,l_nStartLine+i,"")
        call type(39,l_nStartLine+i,"")
        //call typeCenter(i+l_nStartLine,sMessage[i],38,false)
        l_sMessage=sMessage[i]
        call typeCenter(i+l_nStartLine,l_sMessage,38,false)
        call type(0,l_nStartLine+i,"│"+l_sMessage+"│")
      endFor
      // end LINE
      call type(0,l_nStartLine+l_nLine+1,"│                                      │")
      call type(0,l_nStartLine+l_nLine+2,"└──────────────────────────────────────┘")
      // release
      if x_nTime==0
        delay(0.1)
      else
        delay(0)
      endIf
    until (clock()-l_nTime)>=x_nTime
    //
    bShowDialog=false
    bUseRefresh=true
  endIf
end

--- type.pgx ---
public program type(num pX (dimensions=1), num pY (dimensions=1), string pStr (dimensions=1))
begin
  //---------------------------------
  //  S H O W   O N E   S T R I N G
  //---------------------------------
  // Display one string to pX column
  // and pY Line
  //
  gotoxy(pX,pY)
  put(pStr)
end

--- typeCenter.pgx ---
public program typeCenter(num x_nY (dimensions=1), string& x_sStr[] (dimensions=1), num x_nLength (dimensions=1), bool x_bShow (dimensions=1))
  local num lX
  local num lLenStr
  local string lStr
  local num i
begin
  //---------------------------------
  //  S H O W   O N E   S T R I N G
  //---------------------------------
  // type one message in center
  // of the userPage
  //
  // See type()
  //
  lLenStr=getDisplayLen(x_sStr)
  if (lLenStr>x_nLength)
    // comprime
    call strlength(x_sStr,x_nLength)
    lX=(40-x_nLength)/2
  else
    // found the median pos
    lX=20-(lLenStr/2)
    lStr=x_sStr
  endIf
  if x_bShow
    // print on the screen
    call type(lX,x_nY,lStr)
  else
    // add empty space to the string
    for i=1 to lX-1
      lStr=" "+lStr
    endFor
    call strfill(lStr,x_nLength,x_sStr)
  endIf
end

--- typeLen.pgx ---
public program typeLen(num pX (dimensions=1), num pY (dimensions=1), string pStr (dimensions=1), num pLen (dimensions=1))
begin
  //---------------------------------
  //  S H O W   O N E   S T R I N G
  //---------------------------------
  // Display one message with the same
  // number of characters.
  //
  //
  // See type()
  //         1234567890123456789012345678901234567890
  call strlength(pStr,pLen)
  call type(pX,pY,pStr)
end

--- typeMenu.pgx ---
public program typeMenu(num pNumber, string pStr)
  local num lStep
  local num lPosY
  local string lStrEmpty
  local num lMaxLen
  local num i
  local string lStr
  local num lPosX
begin
  //---------------------------------
  //  S H O W   O N E   S T R I N G
  //---------------------------------
  // Display one message in the
  // user menu page
  // 4 characters and 1 space
  //
  //
  lStep=5
  lPosY=13
  lStrEmpty="     "
  if (pNumber>=1) and (pNumber<=8)
    lMaxLen=4
    // Control the len
    // europe case
    if (getDisplayLen(pStr)>lMaxLen)
      if len(pStr)==getDisplayLen(pStr)
        i=find(pStr," ")
        if i<5 and i>2
          lStr=mid(pStr,i,0)
        else
          lStr=mid(pStr,lMaxLen-1,0)
          lStr=lStr+"."
        endIf
      else
        // asia one
        lStr=mid(pStr,2,0)
      endIf
    else
      lStr=pStr
    endIf
    // Position X
    lPosX=(pNumber-1)*lStep+1
    // log
    call strfill(lStr,4,lStr)
    call type(lPosX,lPosY,lStr)
  endIf
end

--- yes_no.pgx ---
public program yes_no(string x_sMessage (dimensions=1), string& x_sYesNo[] (dimensions=1), bool& x_bResult[] (dimensions=1))
  local num i
  local string l_sButton[2]
begin
  //
  // write a yes no question dialog
  //
  if x_sYesNo!=""
    l_sButton[0]=x_sYesNo
  else
    l_sButton[0]="Yes"
  endIf
  //
  if x_sYesNo[1]!=""
    l_sButton[1]=x_sYesNo[1]
  else
    l_sButton[1]="No"
  endIf
  // question Dialog
  call questionDialog(x_sMessage,l_sButton,i)
  // press F8->YES or ENTER
  if i==1 or i==0
    x_bResult=true
  else
    // press escape or F7->NO
    x_bResult=false
  endIf
end

--- yes_no_cancel.pgx ---
public program yes_no_cancel(string x_sMessage (dimensions=1), string& x_sYesNo[] (dimensions=1), bool& x_bResult[] (dimensions=1), bool& x_bCancel[] (dimensions=1))
  local num i
  local string l_sButton[3]
begin
  // INIT
  x_bCancel=false
  l_sButton[0]=x_sYesNo
  l_sButton[1]=x_sYesNo[1]
  l_sButton[2]="Esc"
  // write a yes no cancel question dialog
  call questionDialog(x_sMessage,l_sButton,i)
  // press F8 or enter
  if i==1 or i==0
    x_bResult=true
  else
    // press escape or F6
    if i==-1 or i==3
      x_bCancel=true
    endIf
    // press F7-no
    x_bResult=false
  endIf
end
